FUNCTION_BLOCK FB_DeleteOldestFile
VAR_INPUT
	i_bStart					:BOOL;
	i_sPathDir					:STRING[300];
	i_sKeyword					:STRING:='*';
	i_MaxNumberFiles			:UINT;
END_VAR
VAR_OUTPUT
	q_bBusy							:BOOL;
	q_bDone							:BOOL;
	q_bError						:BOOL;
	q_sOldestFile					:STRING;
	q_iNumberOfFiles				:UINT;
	
END_VAR
VAR
	fbFindFile				:FB_EnumFindFileEntry;
	eCmd					:E_EnumCmdType;
	bExecute				:BOOL;
	stFindFile				:ST_FindFileEntry;
	fbFileDelete			:FB_FileDelete;
	iStep					:INT:=0;
	sPath					:STRING[300];
	bDelete					:BOOL;
	sDeletePath				:STRING[300];
END_VAR

sPath:=CONCAT(i_sPathDir,i_sKeyword);
ACT_Files();
CASE iStep OF
	0:
		q_bBusy:=FALSE;
		IF i_bStart THEN
			q_iNumberOfFiles:=0;
			q_bDone:=FALSE;
			q_bError:=FALSE;
			q_bBusy:=TRUE;
			iStep:=10;
		END_IF
		
	10:
		eCmd := 0;
		bExecute:=TRUE;
		IF fbFindFile.bBusy THEN
			iStep:=20;
		END_IF
		
	20:
		IF NOT fbFindFile.bBusy THEN
			IF NOT fbFindFile.bError AND NOT fbFindFile.bEOE THEN
				q_sOldestFile:=stFindFile.sFileName;
				bExecute:=FALSE;
				iStep:=30;
			ELSIF NOT fbFindFile.bError AND fbFindFile.bEOE THEN
				bExecute:=FALSE;
				iStep:=100;
			ELSIF fbFindFile.bError THEN
				iStep:=999;
			END_IF
		END_IF
		
	30:
		q_iNumberOfFiles:=q_iNumberOfFiles+1;
		iStep:=40;
	
	40:
		eCmd := 1;
		bExecute:=TRUE;
		IF fbFindFile.bBusy THEN
			iStep:=50;
		END_IF
	
	50:
		IF NOT fbFindFile.bBusy THEN
			IF NOT fbFindFile.bError AND NOT fbFindFile.bEOE THEN
				bExecute:=FALSE;
				iStep:=30;
			ELSIF NOT fbFindFile.bError AND fbFindFile.bEOE THEN
				bExecute:=FALSE;
				iStep:=100;
			ELSIF fbFindFile.bError THEN
				iStep:=999;
			END_IF
		END_IF
		
	100:
		eCmd:=2;
		bExecute:=TRUE;
		IF NOT fbFindFile.bBusy THEN
			iStep:=150;
		END_IF
		
	150:
		IF q_iNumberOfFiles >= i_MaxNumberFiles THEN
			iStep:=200;
		ELSE
			iStep:=300;
		END_IF
		
	200:
		sDeletePath:=CONCAT(i_sPathDir,q_sOldestFile);
		bDelete:=TRUE;
		iStep:=210;
	
	210:
		IF NOT fbFileDelete.bBusy THEN
			iStep:=300;
		END_IF
		
	300:
		q_bDone:=TRUE;
		iStep:=0;
		
	999:
		q_bError:=TRUE;
		iStep:=0;
		
		
END_CASE

ACTION ACT_Files:
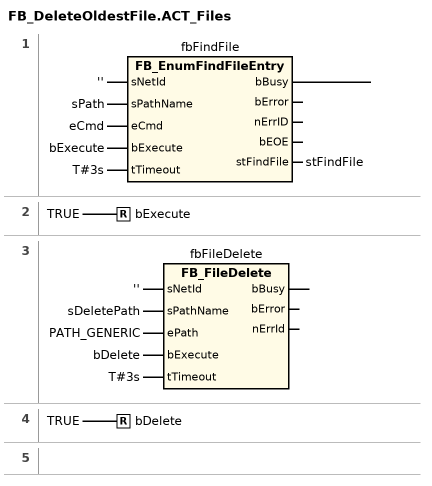
// NETWORK 1
fbFindFile(
    sNetId := '',
    sPathName := sPath,
    eCmd := eCmd,
    bExecute := bExecute,
    tTimeout := T#3s,
    stFindFile => stFindFile); // FB_EnumFindFileEntry

// NETWORK 2
bExecute R= TRUE;

// NETWORK 3
fbFileDelete(
    sNetId := '',
    sPathName := sDeletePath,
    ePath := PATH_GENERIC,
    bExecute := bDelete,
    tTimeout := T#3s); // FB_FileDelete

// NETWORK 4
bDelete R= TRUE;

// NETWORK 5
END_ACTION

END_FUNCTION_BLOCK

(* stored: Version 1.1.0.1, ProductVersion 3.1.4024.12
   POU FB_DeleteOldestFile: Id {4ef72b8d-e6a9-47cb-98b8-b0d83cc2d785}, SpecialFunc None
   Action ACT_Files: Id {935e4c15-c973-4b63-8e3f-58e2c10fbbc4} *)
